{attribute 'qualified_only'}
{attribute 'analysis' := '-33'}
VAR_GLOBAL
	{attribute 'OPC.UA.DA' := '1'}
	MonitorTestData		: MonitorTest;
	{attribute 'OPC.UA.DA' := '1'}
	ReadTestData		: ReadTest;
	{attribute 'OPC.UA.DA' := '1'}
	SymbolTestData		: SymbolTest;
	{attribute 'OPC.UA.DA' := '1'}
	WriteTestData		: WriteTest;
END_VAR

(* stored: Version 1.1.0.1, ProductVersion 3.1.4024.12
   GVL Opc: Id {bcbee6ff-468d-4de1-b7a3-a065b49ecba3} *)
